PROGRAM P_ReadSensors
VAR
	
	readAcc : FB_ReadAccelerometer;
	readGeo : FB_ReadGeophone;
	
	accX : LREAL;
	accY : LREAL;
	accZ : LREAL;
	
	velX : LREAL;
	velY : LREAL;
	velZ : LREAL;
END_VAR

readAcc(accX => accX, accY => accY, accZ => accZ);
readGeo(velX => velX, velY => velY, velZ => velZ);

END_PROGRAM

(* stored: Version 1.1.0.1, ProductVersion 3.1.4024.13
   POU P_ReadSensors: Id {5db38278-0676-4eeb-ab89-3aec0fb96e5a}, SpecialFunc None *)
